// TIA Portal V16 export
// export: Created 2021-11-12T13:31:12.525558Z, ExportSetting WithDefaults, DisplayName Totally Integrated Automation Portal, DisplayVersion V16 Update 3, DisplayName TIA Portal Version Control Interface, DisplayVersion V16 Update 2, DisplayName TIA Portal Openness, DisplayVersion V16 Update 3, DisplayName SINAMICS Startdrive Advanced, DisplayVersion V16 Update 5, DisplayName SINAMICS Startdrive G130, G150, S120, S150, SINAMICS MV, S210, DisplayVersion V16 Update 5, DisplayName SINAMICS Startdrive G110M, G120, G120C, G120D, G120P, G115D, DisplayVersion V16 Update 5, DisplayName STEP 7 Professional, DisplayVersion V16 Update 3, DisplayName STEP 7 Safety, DisplayVersion V16, DisplayName WinCC UA Professional, DisplayVersion V16 Update 3
FUNCTION "Sfty_Interface" : Void   // FC22, F_LAD
{ S7_Optimized_Access := 'TRUE' }
VERSION : 0.1
// Interface from standard program to safety program
// stored: AutoNumber true, IsIECCheckEnabled false, UDAEnableTagReadback false
BEGIN

REGION Network 1: Commisioning signal datab blocks copy
   // Group01 - zone 100 buttons included panel 000-UH11, panel 000-UH10
   // Group02 - zone 200 buttons included panel 000-UH11, panel 000-UH10
   // Group03 - zone 300 buttons included panel 000-UH11, panel 000-UH10
   // Group04 - zone 400 buttons included panel 000-UH11, panel 000-UH10
   // Group05 - panel 000-UH11, panel 000-UH10
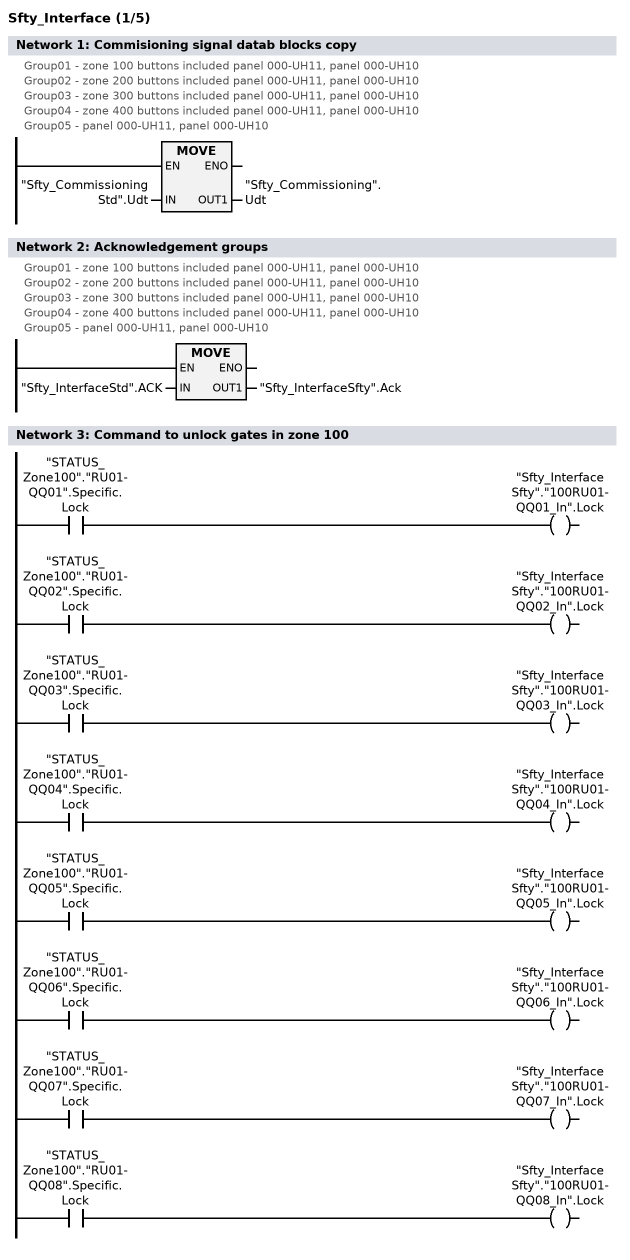
   RUNG wire#powerrail
      { S7_GenerateENO := "TRUE" } Move(in := "Sfty_CommissioningStd".Udt, out1 => "Sfty_Commissioning".Udt)
   END_RUNG
   // the same network as SCL:
   "Sfty_Commissioning".Udt := "Sfty_CommissioningStd".Udt;
END_REGION

REGION Network 2: Acknowledgement groups
   // Group01 - zone 100 buttons included panel 000-UH11, panel 000-UH10
   // Group02 - zone 200 buttons included panel 000-UH11, panel 000-UH10
   // Group03 - zone 300 buttons included panel 000-UH11, panel 000-UH10
   // Group04 - zone 400 buttons included panel 000-UH11, panel 000-UH10
   // Group05 - panel 000-UH11, panel 000-UH10
   RUNG wire#powerrail
      { S7_GenerateENO := "TRUE" } Move(in := "Sfty_InterfaceStd".ACK, out1 => "Sfty_InterfaceSfty".Ack)
   END_RUNG
   // the same network as SCL:
   "Sfty_InterfaceSfty".Ack := "Sfty_InterfaceStd".ACK;
END_REGION

REGION Network 3: Command to unlock gates in zone 100
   RUNG wire#powerrail
      Contact( "STATUS_Zone100"."RU01-QQ01".Specific.Lock )
      Coil( "Sfty_InterfaceSfty"."100RU01-QQ01_In".Lock )
   END_RUNG
   RUNG wire#powerrail
      Contact( "STATUS_Zone100"."RU01-QQ02".Specific.Lock )
      Coil( "Sfty_InterfaceSfty"."100RU01-QQ02_In".Lock )
   END_RUNG
   RUNG wire#powerrail
      Contact( "STATUS_Zone100"."RU01-QQ03".Specific.Lock )
      Coil( "Sfty_InterfaceSfty"."100RU01-QQ03_In".Lock )
   END_RUNG
   RUNG wire#powerrail
      Contact( "STATUS_Zone100"."RU01-QQ04".Specific.Lock )
      Coil( "Sfty_InterfaceSfty"."100RU01-QQ04_In".Lock )
   END_RUNG
   RUNG wire#powerrail
      Contact( "STATUS_Zone100"."RU01-QQ05".Specific.Lock )
      Coil( "Sfty_InterfaceSfty"."100RU01-QQ05_In".Lock )
   END_RUNG
   RUNG wire#powerrail
      Contact( "STATUS_Zone100"."RU01-QQ06".Specific.Lock )
      Coil( "Sfty_InterfaceSfty"."100RU01-QQ06_In".Lock )
   END_RUNG
   RUNG wire#powerrail
      Contact( "STATUS_Zone100"."RU01-QQ07".Specific.Lock )
      Coil( "Sfty_InterfaceSfty"."100RU01-QQ07_In".Lock )
   END_RUNG
   RUNG wire#powerrail
      Contact( "STATUS_Zone100"."RU01-QQ08".Specific.Lock )
      Coil( "Sfty_InterfaceSfty"."100RU01-QQ08_In".Lock )
   END_RUNG
   // the same network as SCL:
   "Sfty_InterfaceSfty"."100RU01-QQ01_In".Lock := "STATUS_Zone100"."RU01-QQ01".Specific.Lock;
   "Sfty_InterfaceSfty"."100RU01-QQ02_In".Lock := "STATUS_Zone100"."RU01-QQ02".Specific.Lock;
   "Sfty_InterfaceSfty"."100RU01-QQ03_In".Lock := "STATUS_Zone100"."RU01-QQ03".Specific.Lock;
   "Sfty_InterfaceSfty"."100RU01-QQ04_In".Lock := "STATUS_Zone100"."RU01-QQ04".Specific.Lock;
   "Sfty_InterfaceSfty"."100RU01-QQ05_In".Lock := "STATUS_Zone100"."RU01-QQ05".Specific.Lock;
   "Sfty_InterfaceSfty"."100RU01-QQ06_In".Lock := "STATUS_Zone100"."RU01-QQ06".Specific.Lock;
   "Sfty_InterfaceSfty"."100RU01-QQ07_In".Lock := "STATUS_Zone100"."RU01-QQ07".Specific.Lock;
   "Sfty_InterfaceSfty"."100RU01-QQ08_In".Lock := "STATUS_Zone100"."RU01-QQ08".Specific.Lock;
END_REGION

REGION Network 4: Command to acknowledge gates in zone 100
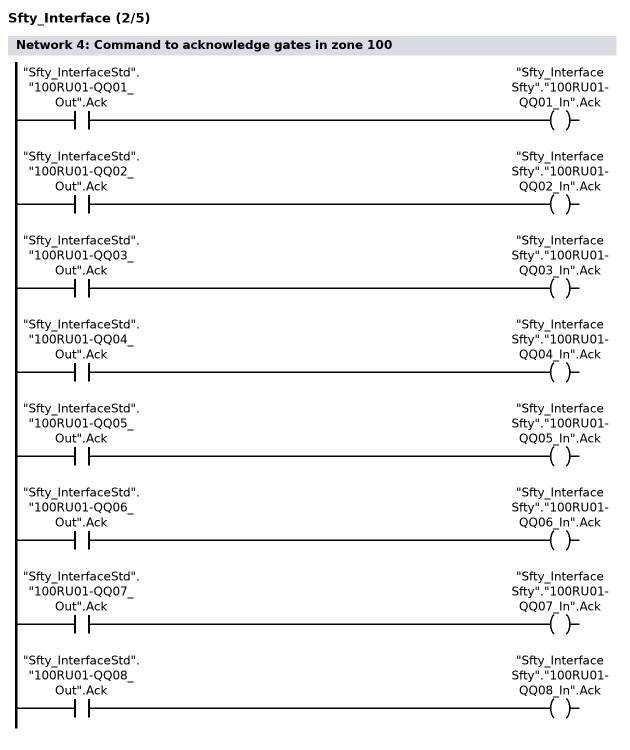
   RUNG wire#powerrail
      Contact( "Sfty_InterfaceStd"."100RU01-QQ01_Out".Ack )
      Coil( "Sfty_InterfaceSfty"."100RU01-QQ01_In".Ack )
   END_RUNG
   RUNG wire#powerrail
      Contact( "Sfty_InterfaceStd"."100RU01-QQ02_Out".Ack )
      Coil( "Sfty_InterfaceSfty"."100RU01-QQ02_In".Ack )
   END_RUNG
   RUNG wire#powerrail
      Contact( "Sfty_InterfaceStd"."100RU01-QQ03_Out".Ack )
      Coil( "Sfty_InterfaceSfty"."100RU01-QQ03_In".Ack )
   END_RUNG
   RUNG wire#powerrail
      Contact( "Sfty_InterfaceStd"."100RU01-QQ04_Out".Ack )
      Coil( "Sfty_InterfaceSfty"."100RU01-QQ04_In".Ack )
   END_RUNG
   RUNG wire#powerrail
      Contact( "Sfty_InterfaceStd"."100RU01-QQ05_Out".Ack )
      Coil( "Sfty_InterfaceSfty"."100RU01-QQ05_In".Ack )
   END_RUNG
   RUNG wire#powerrail
      Contact( "Sfty_InterfaceStd"."100RU01-QQ06_Out".Ack )
      Coil( "Sfty_InterfaceSfty"."100RU01-QQ06_In".Ack )
   END_RUNG
   RUNG wire#powerrail
      Contact( "Sfty_InterfaceStd"."100RU01-QQ07_Out".Ack )
      Coil( "Sfty_InterfaceSfty"."100RU01-QQ07_In".Ack )
   END_RUNG
   RUNG wire#powerrail
      Contact( "Sfty_InterfaceStd"."100RU01-QQ08_Out".Ack )
      Coil( "Sfty_InterfaceSfty"."100RU01-QQ08_In".Ack )
   END_RUNG
   // the same network as SCL:
   "Sfty_InterfaceSfty"."100RU01-QQ01_In".Ack := "Sfty_InterfaceStd"."100RU01-QQ01_Out".Ack;
   "Sfty_InterfaceSfty"."100RU01-QQ02_In".Ack := "Sfty_InterfaceStd"."100RU01-QQ02_Out".Ack;
   "Sfty_InterfaceSfty"."100RU01-QQ03_In".Ack := "Sfty_InterfaceStd"."100RU01-QQ03_Out".Ack;
   "Sfty_InterfaceSfty"."100RU01-QQ04_In".Ack := "Sfty_InterfaceStd"."100RU01-QQ04_Out".Ack;
   "Sfty_InterfaceSfty"."100RU01-QQ05_In".Ack := "Sfty_InterfaceStd"."100RU01-QQ05_Out".Ack;
   "Sfty_InterfaceSfty"."100RU01-QQ06_In".Ack := "Sfty_InterfaceStd"."100RU01-QQ06_Out".Ack;
   "Sfty_InterfaceSfty"."100RU01-QQ07_In".Ack := "Sfty_InterfaceStd"."100RU01-QQ07_Out".Ack;
   "Sfty_InterfaceSfty"."100RU01-QQ08_In".Ack := "Sfty_InterfaceStd"."100RU01-QQ08_Out".Ack;
END_REGION

REGION Network 5: Request to acknowledge closed gate zone 100
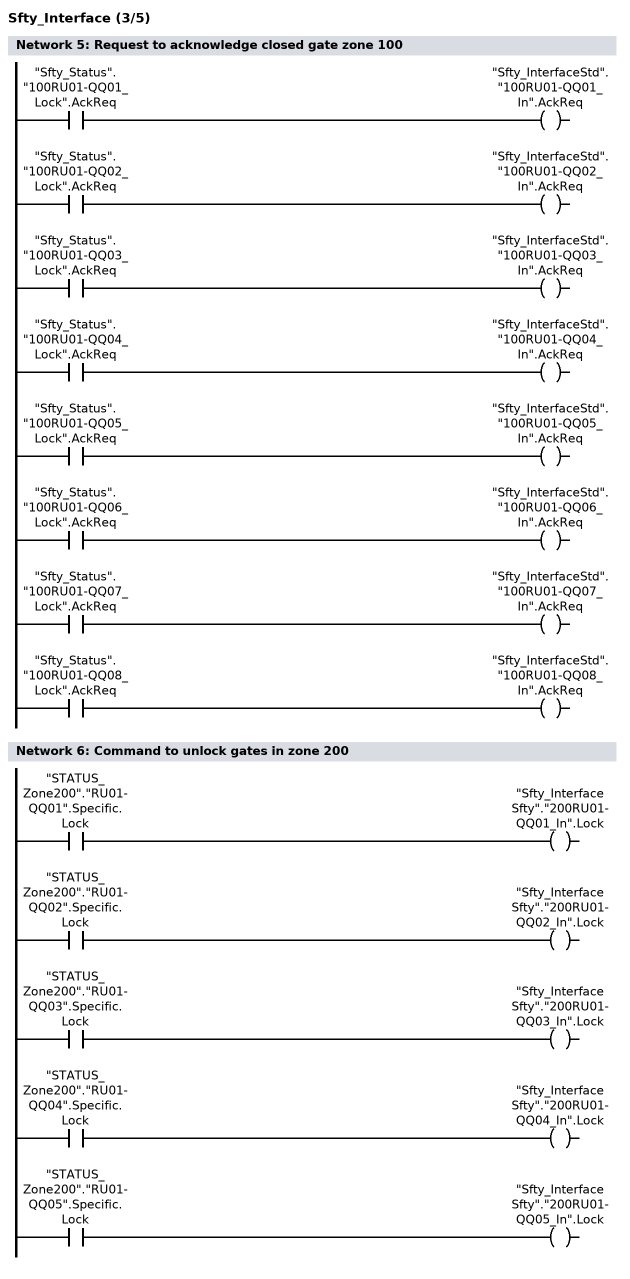
   RUNG wire#powerrail
      Contact( "Sfty_Status"."100RU01-QQ01_Lock".AckReq )
      Coil( "Sfty_InterfaceStd"."100RU01-QQ01_In".AckReq )
   END_RUNG
   RUNG wire#powerrail
      Contact( "Sfty_Status"."100RU01-QQ02_Lock".AckReq )
      Coil( "Sfty_InterfaceStd"."100RU01-QQ02_In".AckReq )
   END_RUNG
   RUNG wire#powerrail
      Contact( "Sfty_Status"."100RU01-QQ03_Lock".AckReq )
      Coil( "Sfty_InterfaceStd"."100RU01-QQ03_In".AckReq )
   END_RUNG
   RUNG wire#powerrail
      Contact( "Sfty_Status"."100RU01-QQ04_Lock".AckReq )
      Coil( "Sfty_InterfaceStd"."100RU01-QQ04_In".AckReq )
   END_RUNG
   RUNG wire#powerrail
      Contact( "Sfty_Status"."100RU01-QQ05_Lock".AckReq )
      Coil( "Sfty_InterfaceStd"."100RU01-QQ05_In".AckReq )
   END_RUNG
   RUNG wire#powerrail
      Contact( "Sfty_Status"."100RU01-QQ06_Lock".AckReq )
      Coil( "Sfty_InterfaceStd"."100RU01-QQ06_In".AckReq )
   END_RUNG
   RUNG wire#powerrail
      Contact( "Sfty_Status"."100RU01-QQ07_Lock".AckReq )
      Coil( "Sfty_InterfaceStd"."100RU01-QQ07_In".AckReq )
   END_RUNG
   RUNG wire#powerrail
      Contact( "Sfty_Status"."100RU01-QQ08_Lock".AckReq )
      Coil( "Sfty_InterfaceStd"."100RU01-QQ08_In".AckReq )
   END_RUNG
   // the same network as SCL:
   "Sfty_InterfaceStd"."100RU01-QQ01_In".AckReq := "Sfty_Status"."100RU01-QQ01_Lock".AckReq;
   "Sfty_InterfaceStd"."100RU01-QQ02_In".AckReq := "Sfty_Status"."100RU01-QQ02_Lock".AckReq;
   "Sfty_InterfaceStd"."100RU01-QQ03_In".AckReq := "Sfty_Status"."100RU01-QQ03_Lock".AckReq;
   "Sfty_InterfaceStd"."100RU01-QQ04_In".AckReq := "Sfty_Status"."100RU01-QQ04_Lock".AckReq;
   "Sfty_InterfaceStd"."100RU01-QQ05_In".AckReq := "Sfty_Status"."100RU01-QQ05_Lock".AckReq;
   "Sfty_InterfaceStd"."100RU01-QQ06_In".AckReq := "Sfty_Status"."100RU01-QQ06_Lock".AckReq;
   "Sfty_InterfaceStd"."100RU01-QQ07_In".AckReq := "Sfty_Status"."100RU01-QQ07_Lock".AckReq;
   "Sfty_InterfaceStd"."100RU01-QQ08_In".AckReq := "Sfty_Status"."100RU01-QQ08_Lock".AckReq;
END_REGION

REGION Network 6: Command to unlock gates in zone 200
   RUNG wire#powerrail
      Contact( "STATUS_Zone200"."RU01-QQ01".Specific.Lock )
      Coil( "Sfty_InterfaceSfty"."200RU01-QQ01_In".Lock )
   END_RUNG
   RUNG wire#powerrail
      Contact( "STATUS_Zone200"."RU01-QQ02".Specific.Lock )
      Coil( "Sfty_InterfaceSfty"."200RU01-QQ02_In".Lock )
   END_RUNG
   RUNG wire#powerrail
      Contact( "STATUS_Zone200"."RU01-QQ03".Specific.Lock )
      Coil( "Sfty_InterfaceSfty"."200RU01-QQ03_In".Lock )
   END_RUNG
   RUNG wire#powerrail
      Contact( "STATUS_Zone200"."RU01-QQ04".Specific.Lock )
      Coil( "Sfty_InterfaceSfty"."200RU01-QQ04_In".Lock )
   END_RUNG
   RUNG wire#powerrail
      Contact( "STATUS_Zone200"."RU01-QQ05".Specific.Lock )
      Coil( "Sfty_InterfaceSfty"."200RU01-QQ05_In".Lock )
   END_RUNG
   // the same network as SCL:
   "Sfty_InterfaceSfty"."200RU01-QQ01_In".Lock := "STATUS_Zone200"."RU01-QQ01".Specific.Lock;
   "Sfty_InterfaceSfty"."200RU01-QQ02_In".Lock := "STATUS_Zone200"."RU01-QQ02".Specific.Lock;
   "Sfty_InterfaceSfty"."200RU01-QQ03_In".Lock := "STATUS_Zone200"."RU01-QQ03".Specific.Lock;
   "Sfty_InterfaceSfty"."200RU01-QQ04_In".Lock := "STATUS_Zone200"."RU01-QQ04".Specific.Lock;
   "Sfty_InterfaceSfty"."200RU01-QQ05_In".Lock := "STATUS_Zone200"."RU01-QQ05".Specific.Lock;
END_REGION

REGION Network 7: Command to acknowledge gates in zone 200
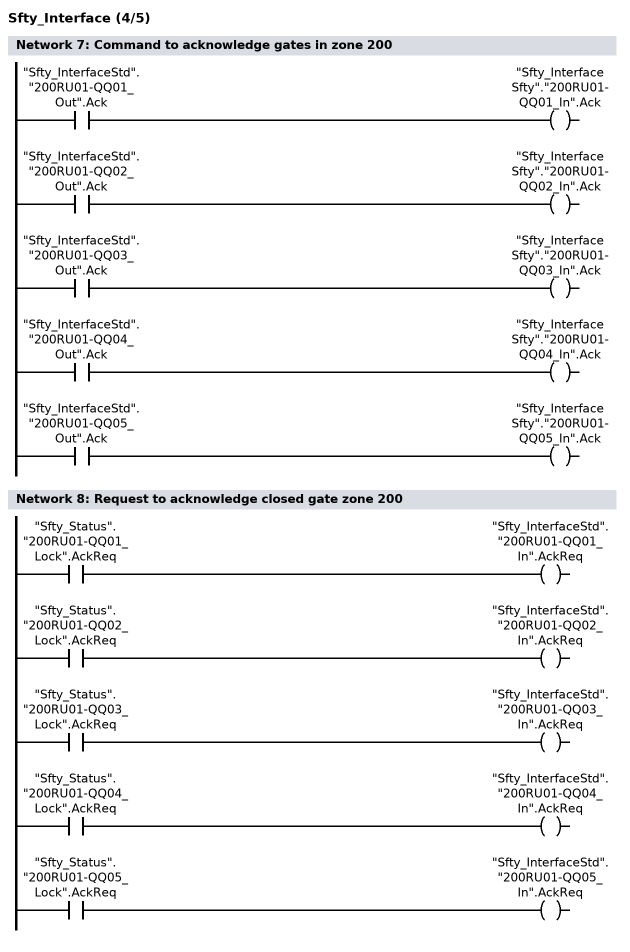
   RUNG wire#powerrail
      Contact( "Sfty_InterfaceStd"."200RU01-QQ01_Out".Ack )
      Coil( "Sfty_InterfaceSfty"."200RU01-QQ01_In".Ack )
   END_RUNG
   RUNG wire#powerrail
      Contact( "Sfty_InterfaceStd"."200RU01-QQ02_Out".Ack )
      Coil( "Sfty_InterfaceSfty"."200RU01-QQ02_In".Ack )
   END_RUNG
   RUNG wire#powerrail
      Contact( "Sfty_InterfaceStd"."200RU01-QQ03_Out".Ack )
      Coil( "Sfty_InterfaceSfty"."200RU01-QQ03_In".Ack )
   END_RUNG
   RUNG wire#powerrail
      Contact( "Sfty_InterfaceStd"."200RU01-QQ04_Out".Ack )
      Coil( "Sfty_InterfaceSfty"."200RU01-QQ04_In".Ack )
   END_RUNG
   RUNG wire#powerrail
      Contact( "Sfty_InterfaceStd"."200RU01-QQ05_Out".Ack )
      Coil( "Sfty_InterfaceSfty"."200RU01-QQ05_In".Ack )
   END_RUNG
   // the same network as SCL:
   "Sfty_InterfaceSfty"."200RU01-QQ01_In".Ack := "Sfty_InterfaceStd"."200RU01-QQ01_Out".Ack;
   "Sfty_InterfaceSfty"."200RU01-QQ02_In".Ack := "Sfty_InterfaceStd"."200RU01-QQ02_Out".Ack;
   "Sfty_InterfaceSfty"."200RU01-QQ03_In".Ack := "Sfty_InterfaceStd"."200RU01-QQ03_Out".Ack;
   "Sfty_InterfaceSfty"."200RU01-QQ04_In".Ack := "Sfty_InterfaceStd"."200RU01-QQ04_Out".Ack;
   "Sfty_InterfaceSfty"."200RU01-QQ05_In".Ack := "Sfty_InterfaceStd"."200RU01-QQ05_Out".Ack;
END_REGION

REGION Network 8: Request to acknowledge closed gate zone 200
   RUNG wire#powerrail
      Contact( "Sfty_Status"."200RU01-QQ01_Lock".AckReq )
      Coil( "Sfty_InterfaceStd"."200RU01-QQ01_In".AckReq )
   END_RUNG
   RUNG wire#powerrail
      Contact( "Sfty_Status"."200RU01-QQ02_Lock".AckReq )
      Coil( "Sfty_InterfaceStd"."200RU01-QQ02_In".AckReq )
   END_RUNG
   RUNG wire#powerrail
      Contact( "Sfty_Status"."200RU01-QQ03_Lock".AckReq )
      Coil( "Sfty_InterfaceStd"."200RU01-QQ03_In".AckReq )
   END_RUNG
   RUNG wire#powerrail
      Contact( "Sfty_Status"."200RU01-QQ04_Lock".AckReq )
      Coil( "Sfty_InterfaceStd"."200RU01-QQ04_In".AckReq )
   END_RUNG
   RUNG wire#powerrail
      Contact( "Sfty_Status"."200RU01-QQ05_Lock".AckReq )
      Coil( "Sfty_InterfaceStd"."200RU01-QQ05_In".AckReq )
   END_RUNG
   // the same network as SCL:
   "Sfty_InterfaceStd"."200RU01-QQ01_In".AckReq := "Sfty_Status"."200RU01-QQ01_Lock".AckReq;
   "Sfty_InterfaceStd"."200RU01-QQ02_In".AckReq := "Sfty_Status"."200RU01-QQ02_Lock".AckReq;
   "Sfty_InterfaceStd"."200RU01-QQ03_In".AckReq := "Sfty_Status"."200RU01-QQ03_Lock".AckReq;
   "Sfty_InterfaceStd"."200RU01-QQ04_In".AckReq := "Sfty_Status"."200RU01-QQ04_Lock".AckReq;
   "Sfty_InterfaceStd"."200RU01-QQ05_In".AckReq := "Sfty_Status"."200RU01-QQ05_Lock".AckReq;
END_REGION

REGION Network 9: AutoStop buttons for robots in zone 100
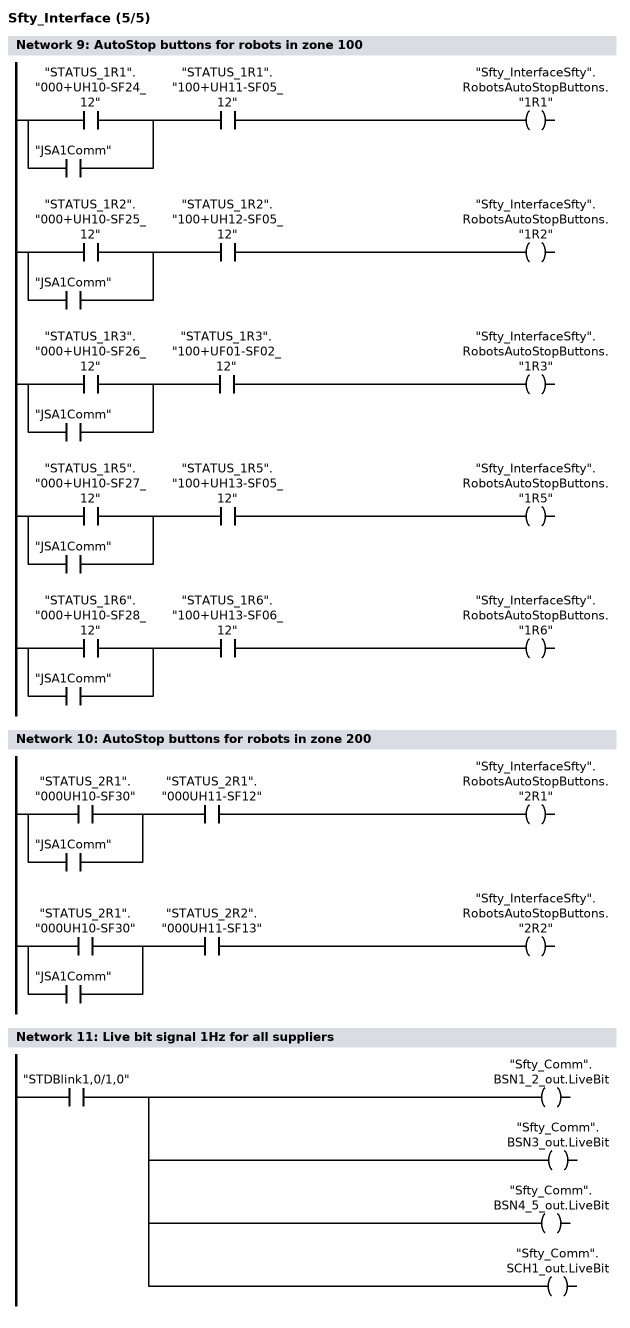
   RUNG wire#powerrail
      Contact( "STATUS_1R1"."000+UH10-SF24_12" )
      wire#w1
      Contact( "STATUS_1R1"."100+UH11-SF05_12" )
      Coil( "Sfty_InterfaceSfty".RobotsAutoStopButtons."1R1" )
   END_RUNG
   RUNG wire#powerrail
      Contact( "JSA1Comm" )
   END_RUNG wire#w1
   RUNG wire#powerrail
      Contact( "STATUS_1R2"."000+UH10-SF25_12" )
      wire#w2
      Contact( "STATUS_1R2"."100+UH12-SF05_12" )
      Coil( "Sfty_InterfaceSfty".RobotsAutoStopButtons."1R2" )
   END_RUNG
   RUNG wire#powerrail
      Contact( "JSA1Comm" )
   END_RUNG wire#w2
   RUNG wire#powerrail
      Contact( "STATUS_1R3"."000+UH10-SF26_12" )
      wire#w3
      Contact( "STATUS_1R3"."100+UF01-SF02_12" )
      Coil( "Sfty_InterfaceSfty".RobotsAutoStopButtons."1R3" )
   END_RUNG
   RUNG wire#powerrail
      Contact( "JSA1Comm" )
   END_RUNG wire#w3
   RUNG wire#powerrail
      Contact( "STATUS_1R5"."000+UH10-SF27_12" )
      wire#w4
      Contact( "STATUS_1R5"."100+UH13-SF05_12" )
      Coil( "Sfty_InterfaceSfty".RobotsAutoStopButtons."1R5" )
   END_RUNG
   RUNG wire#powerrail
      Contact( "JSA1Comm" )
   END_RUNG wire#w4
   RUNG wire#powerrail
      Contact( "STATUS_1R6"."000+UH10-SF28_12" )
      wire#w5
      Contact( "STATUS_1R6"."100+UH13-SF06_12" )
      Coil( "Sfty_InterfaceSfty".RobotsAutoStopButtons."1R6" )
   END_RUNG
   RUNG wire#powerrail
      Contact( "JSA1Comm" )
   END_RUNG wire#w5
   // the same network as SCL:
   "Sfty_InterfaceSfty".RobotsAutoStopButtons."1R1" := ("STATUS_1R1"."000+UH10-SF24_12" OR "JSA1Comm") AND "STATUS_1R1"."100+UH11-SF05_12";
   "Sfty_InterfaceSfty".RobotsAutoStopButtons."1R2" := ("STATUS_1R2"."000+UH10-SF25_12" OR "JSA1Comm") AND "STATUS_1R2"."100+UH12-SF05_12";
   "Sfty_InterfaceSfty".RobotsAutoStopButtons."1R3" := ("STATUS_1R3"."000+UH10-SF26_12" OR "JSA1Comm") AND "STATUS_1R3"."100+UF01-SF02_12";
   "Sfty_InterfaceSfty".RobotsAutoStopButtons."1R5" := ("STATUS_1R5"."000+UH10-SF27_12" OR "JSA1Comm") AND "STATUS_1R5"."100+UH13-SF05_12";
   "Sfty_InterfaceSfty".RobotsAutoStopButtons."1R6" := ("STATUS_1R6"."000+UH10-SF28_12" OR "JSA1Comm") AND "STATUS_1R6"."100+UH13-SF06_12";
END_REGION

REGION Network 10: AutoStop buttons for robots in zone 200
   RUNG wire#powerrail
      Contact( "STATUS_2R1"."000UH10-SF30" )
      wire#w1
      Contact( "STATUS_2R1"."000UH11-SF12" )
      Coil( "Sfty_InterfaceSfty".RobotsAutoStopButtons."2R1" )
   END_RUNG
   RUNG wire#powerrail
      Contact( "JSA1Comm" )
   END_RUNG wire#w1
   RUNG wire#powerrail
      Contact( "STATUS_2R1"."000UH10-SF30" )
      wire#w2
      Contact( "STATUS_2R2"."000UH11-SF13" )
      Coil( "Sfty_InterfaceSfty".RobotsAutoStopButtons."2R2" )
   END_RUNG
   RUNG wire#powerrail
      Contact( "JSA1Comm" )
   END_RUNG wire#w2
   // the same network as SCL:
   "Sfty_InterfaceSfty".RobotsAutoStopButtons."2R1" := ("STATUS_2R1"."000UH10-SF30" OR "JSA1Comm") AND "STATUS_2R1"."000UH11-SF12";
   "Sfty_InterfaceSfty".RobotsAutoStopButtons."2R2" := ("STATUS_2R1"."000UH10-SF30" OR "JSA1Comm") AND "STATUS_2R2"."000UH11-SF13";
END_REGION

REGION Network 11: Live bit signal 1Hz for all suppliers
   RUNG wire#powerrail
      Contact( "STDBlink1,0/1,0" )
      wire#w1
      Coil( "Sfty_Comm".BSN1_2_out.LiveBit )
   END_RUNG
   RUNG wire#w1
      Coil( "Sfty_Comm".BSN3_out.LiveBit )
   END_RUNG
   RUNG wire#w1
      Coil( "Sfty_Comm".BSN4_5_out.LiveBit )
   END_RUNG
   RUNG wire#w1
      Coil( "Sfty_Comm".SCH1_out.LiveBit )
   END_RUNG
   // the same network as SCL:
   "Sfty_Comm".BSN1_2_out.LiveBit := "STDBlink1,0/1,0";
   "Sfty_Comm".BSN3_out.LiveBit := "STDBlink1,0/1,0";
   "Sfty_Comm".BSN4_5_out.LiveBit := "STDBlink1,0/1,0";
   "Sfty_Comm".SCH1_out.LiveBit := "STDBlink1,0/1,0";
END_REGION
END_FUNCTION
